Staubli VAL3: actMovement.pgx

program actMovement()
begin
  putln("actMovement called")
  putln(sInput)

end
